// TIA Portal V19 export
TYPE "HEADER"
   STRUCT
      REQ_REF : Byte;
      REQ_ID : Byte;
      AXIS : Byte;
      NO_PARAM : Byte;
   END_STRUCT;
END_TYPE
